              global tcp= get_actual_tcp_pose ()
              $ 1343 "offset_altura≔p[tcp[0],tcp[1],((alta-0.0095)-(acomodo/1000)),tcp[3],tcp[4],tcp[5]]"
              global offset_altura=p[tcp[0],tcp[1],((alta-0.0095)-(acomodo/1000)),tcp[3],tcp[4],tcp[5]]
              $ 1344 "MoveL"
              $ 1345 "offset_altura" "breakAfter"
              movel(offset_altura, a=0.04, v=0.03)
            end
            $ 1346 "Freemove"
            $ 1347 "Wait: 2.0"
            sleep(2.0)
            $ 1348 "freedrive_mode()"
            freedrive_mode()
            $ 1349 "Wait: 2.5"
            sleep(2.5)
            $ 1350 "end_freedrive_mode()"
            end_freedrive_mode()
            $ 1351 "Wait: 0.3"
            sleep(0.3)
            $ 1352 "Set CO[1]=Encender"
            set_configurable_digital_out(1, True)
            $ 1353 "Wait: 1.0"
            sleep(1.0)
            $ 1354 "Wait: 0.3"
            sleep(0.3)
            $ 1355 "Wait: 0.3"
            sleep(0.3)
            $ 1356 "Wait: 0.3"
            sleep(0.3)
            $ 1357 "Loop 2 times"
            Loop_50 = 0
            while (Loop_50 < 2):
              $ 1358 "Poses_taladrado≔pose_sub(get_actual_tcp_pose(), bajada_broca)"
              global Poses_taladrado= pose_sub ( get_actual_tcp_pose (), bajada_broca)
              $ 1359 "Poses_taladrado" "breakAfter"
              movel(Poses_taladrado, a=0.005, v=0.001)
              $ 1360 "If bajada_broca≟p[0,0,0.018,0,0,0]"
              if (bajada_broca == p[0,0,0.018,0,0,0]):
                $ 1361 "num_barreno≔str_cat('Barreno: ',barrenoActual)"
                global num_barreno=str_cat("Barreno: ",barrenoActual)
                $ 1362 "tcp_actual≔get_actual_tcp_pose()"
                global tcp_actual= get_actual_tcp_pose ()
                $ 1363 "X_actual≔str_cat('     X: ',tcp_actual[0])"
                global X_actual=str_cat("     X: ",tcp_actual[0])
                $ 1364 "Y_actual≔str_cat('     Y: ',tcp_actual[1])"
                global Y_actual=str_cat("     Y: ",tcp_actual[1])
                $ 1365 "pos_barreno≔str_cat(X_actual,Y_actual)"
                global pos_barreno=str_cat(X_actual,Y_actual)
                $ 1366 "textmsg(num_barreno,pos_barreno)"
                textmsg(num_barreno,pos_barreno)
              end
              $ 1367 "Poses_taladrado≔pose_add(get_actual_tcp_pose(), bajada_broca)"
              global Poses_taladrado= pose_add ( get_actual_tcp_pose (), bajada_broca)
              $ 1368 "Poses_taladrado" "breakAfter"
              movel(Poses_taladrado, a=0.01, v=0.01)
              $ 1369 "bajada_broca≔pose_add(bajada_broca, p[0,0,0.009,0,0,0])"
              global bajada_broca= pose_add (bajada_broca, p[0,0,0.009,0,0,0])
              Loop_50 = Loop_50 + 1
            end
            $ 1370 "Direction: Base Z+"
            global move_thread_flag_1370=0
            thread move_thread_1370():
              enter_critical
              move_thread_flag_1370 = 1
              local towardsPos=calculate_point_to_move_towards(p[0.0,0.0,0.0,0.0,0.0,0.0], [0.0,0.0,1.0], 0.05)
              movel(towardsPos, a=0.01, v=0.01)
              move_thread_flag_1370 = 2
              exit_critical
            end
            move_thread_flag_1370 = 0
            move_thread_han_1370 = run move_thread_1370()
            while (True):
              sleep(1.0E-10)
              if (move_thread_flag_1370 > 1):
                join move_thread_han_1370
                $ 1371 "Until (distance)"
                break
              end
              sync()
            end
            $ 1372 "MoveJ"
            $ 1373 "internos" "breakAfter"
            movej(internos, a=0.6981317007977318, v=0.5235987755982988)
            $ 1374 "Wait: 0.3"
            sleep(0.3)
            $ 1375 "Set CO[1]=Apagar"
            set_configurable_digital_out(1, False)
            $ 1376 "Wait: 0.3"
            sleep(0.3)
            $ 1377 "If barrenoActual≟13 or barrenoActual≟27"
            if (barrenoActual == 13  or  barrenoActual == 27):
              $ 1378 "Direction: Base Z+"
              global move_thread_flag_1378=0
              thread move_thread_1378():
                enter_critical
                move_thread_flag_1378 = 1
                local towardsPos=calculate_point_to_move_towards(p[0.0,0.0,0.0,0.0,0.0,0.0], [0.0,0.0,1.0], 0.03)
                movel(towardsPos, a=0.04, v=0.03)
                move_thread_flag_1378 = 2
                exit_critical
              end
              move_thread_flag_1378 = 0
              move_thread_han_1378 = run move_thread_1378()
              while (True):
                sleep(1.0E-10)
                if (move_thread_flag_1378 > 1):
                  join move_thread_han_1378
                  $ 1379 "Until (distance)"
                  break
                end
                sync()
              end
              $ 1380 "MoveJ"
              $ 1381 "Zona_der1" "breakAfter"
              movej(get_inverse_kin(Zona_der1_p, qnear=Zona_der1_q), a=0.6981317007977318, v=0.5235987755982988)
              $ 1382 "Posicion_Cero" "breakAfter"
              movej(get_inverse_kin(Posicion_Cero_p, qnear=Posicion_Cero_q), a=0.6981317007977318, v=0.5235987755982988)
              $ 1383 "Call Quitar_Broca_Chida"
              Quitar_Broca_Chida()
              $ 1384 "If barrenoActual≟13"
              if (barrenoActual == 13):
                $ 1385 "Call Poner_Broca"
                Poner_Broca()
              else:
                $ 1386 "ElseIf barrenoActual≟27"
                if (barrenoActual == 27):
                  $ 1387 "Call Poner_Broca"
                  Poner_Broca()
                end
              end
              $ 1388 "MoveJ"
              $ 1389 "Posicion_Cero" "breakAfter"
              movej(get_inverse_kin(Posicion_Cero_p, qnear=Posicion_Cero_q), a=0.6981317007977318, v=0.5235987755982988)
              $ 1390 "Zona_der1" "breakAfter"
              movej(get_inverse_kin(Zona_der1_p, qnear=Zona_der1_q), a=0.6981317007977318, v=0.5235987755982988)
            end
            $ 1391 "barrenoActual≔barrenoActual+1"
            global barrenoActual=barrenoActual+1
          end
          $ 1392 "Linea 2 a 1935"
          $ 1393 "broca≔1935"
          global broca=1935
          $ 1394 "Buje_inicial"
          $ 1395 "Buje_Inicial≔L2B2"
          global Buje_Inicial=L2B2
          $ 1396 "Buje_final"
          $ 1397 "Buje_Final≔L2B1"
          global Buje_Final=L2B1
          $ 1398 "barrenosTotales≔27"
          global barrenosTotales=27
          $ 1399 "barrenoActual≔1"
          global barrenoActual=1
          $ 1400 "Loop barrenoActual≤barrenosTotales"
          while (barrenoActual <= barrenosTotales):
            $ 1401 "MoveL"
            $ 1402 "bajada_broca≔p[0,0,0.009,0,0,0]"
            global bajada_broca=p[0,0,0.009,0,0,0]
            $ 1403 "internos≔interpolate_pose(Buje_Inicial, Buje_Final, ((barrenoActual)-1)/((barrenosTotales)-1))"
            global internos= interpolate_pose (Buje_Inicial, Buje_Final, ((barrenoActual)-1)/((barrenosTotales)-1))
            $ 1404 "Alturas"
            $ 1405 "If barrenoActual≟1 or barrenoActual≟3 or barrenoActual≟5 or barrenoActual≟7 or barrenoActual≟9 or barrenoActual≟11 or barrenoActual≟13 or barrenoActual≟15 or barrenoActual≟17 or barrenoActual≟19 or barrenoActual≟21 or barrenoActual≟23 or barrenoActual≟25 or barrenoActual≟27"
            if (barrenoActual == 1  or  barrenoActual == 3  or  barrenoActual == 5  or  barrenoActual == 7  or  barrenoActual == 9  or  barrenoActual == 11  or  barrenoActual == 13  or  barrenoActual == 15  or  barrenoActual == 17  or  barrenoActual == 19  or  barrenoActual == 21  or  barrenoActual == 23  or  barrenoActual == 25  or  barrenoActual == 27):
              $ 1406 "Set mensaje_mw10=200"
              modbus_set_output_register("mensaje_mw10", 200)
              $ 1407 "Wait Continuar_M30=HI"
              while (modbus_get_signal_status("Continuar_M30") == False):
                sync()
              end
              $ 1408 "Wait: 1.0"
              sleep(1.0)
              $ 1409 "Set mensaje_mw10=150"
              modbus_set_output_register("mensaje_mw10", 150)
              $ 1410 "Wait: 1.0"
              sleep(1.0)
            end
            $ 1411 "MoveJ"
            $ 1412 "internos" "breakAfter"
            movej(internos, a=0.6981317007977318, v=0.5235987755982988)
            $ 1413 "Wait: 2.0"
            sleep(2.0)
            $ 1414 "If P1h[2]<P2h[2]"
            if (P1h[2]<P2h[2]):
              $ 1415 "acomodo≔(altura/(barrenosTotales-1))*(barrenoActual-1)"
              global acomodo=(altura/(barrenosTotales-1))*(barrenoActual-1)
              $ 1416 "tcp≔get_actual_tcp_pose()"
              global tcp= get_actual_tcp_pose ()
              $ 1417 "offset_altura≔p[tcp[0],tcp[1],((alta-0.0095)-(acomodo/1000)),tcp[3],tcp[4],tcp[5]]"
              global offset_altura=p[tcp[0],tcp[1],((alta-0.0095)-(acomodo/1000)),tcp[3],tcp[4],tcp[5]]
              $ 1418 "MoveL"
              $ 1419 "offset_altura" "breakAfter"
              movel(offset_altura, a=0.04, v=0.03)
            else:
              $ 1420 "Else" "noBreak"
              $ 1421 "acomodo≔(altura/(barrenosTotales-1))*(26-(barrenoActual-1))"
              global acomodo=(altura/(barrenosTotales-1))*(26-(barrenoActual-1))
              $ 1422 "tcp≔get_actual_tcp_pose()"
              global tcp= get_actual_tcp_pose ()
              $ 1423 "offset_altura≔p[tcp[0],tcp[1],((alta-0.0095)-(acomodo/1000)),tcp[3],tcp[4],tcp[5]]"
              global offset_altura=p[tcp[0],tcp[1],((alta-0.0095)-(acomodo/1000)),tcp[3],tcp[4],tcp[5]]
              $ 1424 "MoveL"
              $ 1425 "offset_altura" "breakAfter"
              movel(offset_altura, a=0.04, v=0.03)
            end
            $ 1426 "Freemove"
            $ 1427 "Wait: 2.0"
            sleep(2.0)
            $ 1428 "freedrive_mode()"
            freedrive_mode()
            $ 1429 "Wait: 2.5"
            sleep(2.5)
            $ 1430 "end_freedrive_mode()"
            end_freedrive_mode()
            $ 1431 "Wait: 0.3"
            sleep(0.3)
            $ 1432 "Set CO[1]=Encender"
            set_configurable_digital_out(1, True)
            $ 1433 "Wait: 1.0"
            sleep(1.0)
            $ 1434 "Wait: 0.3"
            sleep(0.3)
            $ 1435 "Wait: 0.3"
            sleep(0.3)
            $ 1436 "Wait: 0.3"
            sleep(0.3)
            $ 1437 "Loop 2 times"
            Loop_54 = 0
            while (Loop_54 < 2):
              $ 1438 "Poses_taladrado≔pose_sub(get_actual_tcp_pose(), bajada_broca)"
              global Poses_taladrado= pose_sub ( get_actual_tcp_pose (), bajada_broca)
              $ 1439 "Poses_taladrado" "breakAfter"
              movel(Poses_taladrado, a=0.005, v=0.001)
              $ 1440 "If bajada_broca≟p[0,0,0.018,0,0,0]"
              if (bajada_broca == p[0,0,0.018,0,0,0]):
                $ 1441 "num_barreno≔str_cat('Barreno: ',barrenoActual)"
                global num_barreno=str_cat("Barreno: ",barrenoActual)
                $ 1442 "tcp_actual≔get_actual_tcp_pose()"
                global tcp_actual= get_actual_tcp_pose ()
                $ 1443 "X_actual≔str_cat('     X: ',tcp_actual[0])"
                global X_actual=str_cat("     X: ",tcp_actual[0])
                $ 1444 "Y_actual≔str_cat('     Y: ',tcp_actual[1])"
                global Y_actual=str_cat("     Y: ",tcp_actual[1])
                $ 1445 "pos_barreno≔str_cat(X_actual,Y_actual)"
                global pos_barreno=str_cat(X_actual,Y_actual)
                $ 1446 "textmsg(num_barreno,pos_barreno)"
                textmsg(num_barreno,pos_barreno)
              end
              $ 1447 "Poses_taladrado≔pose_add(get_actual_tcp_pose(), bajada_broca)"
              global Poses_taladrado= pose_add ( get_actual_tcp_pose (), bajada_broca)
              $ 1448 "Poses_taladrado" "breakAfter"
              movel(Poses_taladrado, a=0.01, v=0.01)
              $ 1449 "bajada_broca≔pose_add(bajada_broca, p[0,0,0.009,0,0,0])"
              global bajada_broca= pose_add (bajada_broca, p[0,0,0.009,0,0,0])
              Loop_54 = Loop_54 + 1
            end
            $ 1450 "Direction: Base Z+"
            global move_thread_flag_1450=0
            thread move_thread_1450():
              enter_critical
              move_thread_flag_1450 = 1
              local towardsPos=calculate_point_to_move_towards(p[0.0,0.0,0.0,0.0,0.0,0.0], [0.0,0.0,1.0], 0.05)
              movel(towardsPos, a=0.01, v=0.01)
              move_thread_flag_1450 = 2
              exit_critical
            end
            move_thread_flag_1450 = 0
            move_thread_han_1450 = run move_thread_1450()
            while (True):
              sleep(1.0E-10)
              if (move_thread_flag_1450 > 1):
                join move_thread_han_1450
                $ 1451 "Until (distance)"
                break
              end
              sync()
            end
            $ 1452 "MoveJ"
            $ 1453 "internos" "breakAfter"
            movej(internos, a=0.6981317007977318, v=0.5235987755982988)
            $ 1454 "Wait: 0.3"
            sleep(0.3)
            $ 1455 "Set CO[1]=Apagar"
            set_configurable_digital_out(1, False)
            $ 1456 "Wait: 0.3"
            sleep(0.3)
            $ 1457 "If barrenoActual≟13"
            if (barrenoActual == 13):
              $ 1458 "Direction: Base Z+"
              global move_thread_flag_1458=0
              thread move_thread_1458():
                enter_critical
                move_thread_flag_1458 = 1
                local towardsPos=calculate_point_to_move_towards(p[0.0,0.0,0.0,0.0,0.0,0.0], [0.0,0.0,1.0], 0.03)
                movel(towardsPos, a=0.04, v=0.03)
                move_thread_flag_1458 = 2
                exit_critical
              end
              move_thread_flag_1458 = 0
              move_thread_han_1458 = run move_thread_1458()
              while (True):
                sleep(1.0E-10)
                if (move_thread_flag_1458 > 1):
                  join move_thread_han_1458
                  $ 1459 "Until (distance)"
                  break
                end
                sync()
              end
              $ 1460 "MoveJ"
              $ 1461 "Zona_der1" "breakAfter"
              movej(get_inverse_kin(Zona_der1_p, qnear=Zona_der1_q), a=1.3962634015954636, v=1.0471975511965976)
              $ 1462 "Posicion_Cero" "breakAfter"
              movej(get_inverse_kin(Posicion_Cero_p, qnear=Posicion_Cero_q), a=1.3962634015954636, v=1.0471975511965976)
              $ 1463 "Call Quitar_Broca_Chida"
              Quitar_Broca_Chida()
              $ 1464 "Call Poner_Broca"
              Poner_Broca()
              $ 1465 "MoveJ"
              $ 1466 "Posicion_Cero" "breakAfter"
              movej(get_inverse_kin(Posicion_Cero_p, qnear=Posicion_Cero_q), a=1.3962634015954636, v=1.0471975511965976)
              $ 1467 "Zona_der1" "breakAfter"
              movej(get_inverse_kin(Zona_der1_p, qnear=Zona_der1_q), a=1.3962634015954636, v=1.0471975511965976)
            else:
              $ 1468 "ElseIf barrenoActual≟27"
              if (barrenoActual == 27):
                $ 1469 "Direction: Base Z+"
                global move_thread_flag_1469=0
                thread move_thread_1469():
                  enter_critical
                  move_thread_flag_1469 = 1
                  local towardsPos=calculate_point_to_move_towards(p[0.0,0.0,0.0,0.0,0.0,0.0], [0.0,0.0,1.0], 0.03)
                  movel(towardsPos, a=0.04, v=0.03)
                  move_thread_flag_1469 = 2
                  exit_critical
                end
                move_thread_flag_1469 = 0
                move_thread_han_1469 = run move_thread_1469()
                while (True):
                  sleep(1.0E-10)
                  if (move_thread_flag_1469 > 1):
                    join move_thread_han_1469
                    $ 1470 "Until (distance)"
                    break
                  end
                  sync()
                end
                $ 1471 "MoveJ"
                $ 1472 "Zona_der1" "breakAfter"
                movej(get_inverse_kin(Zona_der1_p, qnear=Zona_der1_q), a=1.3962634015954636, v=1.0471975511965976)
                $ 1473 "Posicion_Cero" "breakAfter"
                movej(get_inverse_kin(Posicion_Cero_p, qnear=Posicion_Cero_q), a=1.3962634015954636, v=1.0471975511965976)
                $ 1474 "Call Quitar_Broca_Chida"
                Quitar_Broca_Chida()
                $ 1475 "Set carrusel_home=Encender"
                modbus_set_output_signal("carrusel_home", True)
                $ 1476 "Wait: 1.0"
                sleep(1.0)
                $ 1477 "Set carrusel_home=Apagar"
                modbus_set_output_signal("carrusel_home", False)
                $ 1478 "Set mensaje_mw10=85"
                modbus_set_output_register("mensaje_mw10", 85)
                $ 1479 "Wait Continuar_M30=HI"
                while (modbus_get_signal_status("Continuar_M30") == False):
                  sync()
                end
                $ 1480 "Wait: 1.0"
                sleep(1.0)
                $ 1481 "Set mensaje_mw10=120"
                modbus_set_output_register("mensaje_mw10", 120)
                $ 1482 "Wait Continuar_M30=HI"
                while (modbus_get_signal_status("Continuar_M30") == False):
                  sync()
                end
                $ 1483 "Wait: 1.0"
                sleep(1.0)
                $ 1484 "Set carrusel_home=Encender"
                modbus_set_output_signal("carrusel_home", True)
                $ 1485 "Wait: 1.0"
                sleep(1.0)
                $ 1486 "Set carrusel_home=Apagar"
                modbus_set_output_signal("carrusel_home", False)
                $ 1487 "Set mensaje_mw10=90"
                modbus_set_output_register("mensaje_mw10", 90)
                $ 1488 "Wait Continuar_M30=HI"
                while (modbus_get_signal_status("Continuar_M30") == False):
                  sync()
                end
                $ 1489 "Wait: 1.0"
                sleep(1.0)
                $ 1490 "Call Poner_Broca"
                Poner_Broca()
                $ 1491 "broca≔217"
                global broca=217
                $ 1492 "MoveJ"
                $ 1493 "Posicion_Cero" "breakAfter"
                movej(get_inverse_kin(Posicion_Cero_p, qnear=Posicion_Cero_q), a=1.3962634015954636, v=1.0471975511965976)
                $ 1494 "Zona_der1" "breakAfter"
                movej(get_inverse_kin(Zona_der1_p, qnear=Zona_der1_q), a=1.3962634015954636, v=1.0471975511965976)
                $ 1495 "Set mensaje_mw10=95"
                modbus_set_output_register("mensaje_mw10", 95)
                $ 1496 "Wait Continuar_M30=HI"
                while (modbus_get_signal_status("Continuar_M30") == False):
                  sync()
                end
                $ 1497 "Wait: 1.0"
                sleep(1.0)
                $ 1498 "Set mensaje_mw10=150"
                modbus_set_output_register("mensaje_mw10", 150)
                $ 1499 "Wait Continuar_M30=HI"
                while (modbus_get_signal_status("Continuar_M30") == False):
                  sync()
                end
                $ 1500 "Wait: 1.0"
                sleep(1.0)
              end
            end
            $ 1501 "barrenoActual≔barrenoActual+1"
            global barrenoActual=barrenoActual+1
          end
          $ 1502 "Linea 1 a 217"
          $ 1503 "broca≔217"
          global broca=217
          $ 1504 "Buje_inicial"
          $ 1505 "Buje_Inicial≔L1B2"
          global Buje_Inicial=L1B2
          $ 1506 "Buje_final"
          $ 1507 "Buje_Final≔L1B1"
          global Buje_Final=L1B1
          $ 1508 "barrenosTotales≔27"
          global barrenosTotales=27
          $ 1509 "barrenoActual≔1"
          global barrenoActual=1
          $ 1510 "Loop barrenoActual≤barrenosTotales"
          while (barrenoActual <= barrenosTotales):
            $ 1511 "MoveL"
            $ 1512 "bajada_broca≔p[0,0,0.018,0,0,0]"
            global bajada_broca=p[0,0,0.018,0,0,0]
            $ 1513 "internos≔interpolate_pose(Buje_Inicial, Buje_Final, ((barrenoActual)-1)/((barrenosTotales)-1))"
            global internos= interpolate_pose (Buje_Inicial, Buje_Final, ((barrenoActual)-1)/((barrenosTotales)-1))
            $ 1514 "Wait: 2.0"
            sleep(2.0)
            $ 1515 "Alturas"
            $ 1516 "If barrenoActual≟1 or barrenoActual≟3 or barrenoActual≟5 or barrenoActual≟7 or barrenoActual≟9 or barrenoActual≟11 or barrenoActual≟13 or barrenoActual≟15 or barrenoActual≟17 or barrenoActual≟19 or barrenoActual≟21 or barrenoActual≟23 or barrenoActual≟25 or barrenoActual≟27"
            if (barrenoActual == 1  or  barrenoActual == 3  or  barrenoActual == 5  or  barrenoActual == 7  or  barrenoActual == 9  or  barrenoActual == 11  or  barrenoActual == 13  or  barrenoActual == 15  or  barrenoActual == 17  or  barrenoActual == 19  or  barrenoActual == 21  or  barrenoActual == 23  or  barrenoActual == 25  or  barrenoActual == 27):
              $ 1517 "Set mensaje_mw10=200"
              modbus_set_output_register("mensaje_mw10", 200)
              $ 1518 "Wait Continuar_M30=HI"
              while (modbus_get_signal_status("Continuar_M30") == False):
                sync()
              end
              $ 1519 "Wait: 1.0"
              sleep(1.0)
              $ 1520 "Set mensaje_mw10=150"
              modbus_set_output_register("mensaje_mw10", 150)
              $ 1521 "Wait: 1.0"
              sleep(1.0)
            end
            $ 1522 "MoveJ"
            $ 1523 "internos" "breakAfter"
            movej(internos, a=0.6981317007977318, v=0.5235987755982988)
            $ 1524 "Wait: 2.0"
            sleep(2.0)
            $ 1525 "If P1h[2]<P2h[2]"
            if (P1h[2]<P2h[2]):
              $ 1526 "acomodo≔(altura/(barrenosTotales-1))*(barrenoActual-1)"
              global acomodo=(altura/(barrenosTotales-1))*(barrenoActual-1)
              $ 1527 "tcp≔get_actual_tcp_pose()"
              global tcp= get_actual_tcp_pose ()
              $ 1528 "offset_altura≔p[tcp[0],tcp[1],((alta-0.0095)-(acomodo/1000)),tcp[3],tcp[4],tcp[5]]"
              global offset_altura=p[tcp[0],tcp[1],((alta-0.0095)-(acomodo/1000)),tcp[3],tcp[4],tcp[5]]
              $ 1529 "MoveL"
              $ 1530 "offset_altura" "breakAfter"
              movel(offset_altura, a=0.04, v=0.03)
            else:
              $ 1531 "Else" "noBreak"
              $ 1532 "acomodo≔(altura/(barrenosTotales-1))*(26-(barrenoActual-1))"
              global acomodo=(altura/(barrenosTotales-1))*(26-(barrenoActual-1))
              $ 1533 "tcp≔get_actual_tcp_pose()"
              global tcp= get_actual_tcp_pose ()
              $ 1534 "offset_altura≔p[tcp[0],tcp[1],((alta-0.0095)-(acomodo/1000)),tcp[3],tcp[4],tcp[5]]"
              global offset_altura=p[tcp[0],tcp[1],((alta-0.0095)-(acomodo/1000)),tcp[3],tcp[4],tcp[5]]
              $ 1535 "MoveL"
              $ 1536 "offset_altura" "breakAfter"
              movel(offset_altura, a=0.04, v=0.03)
            end
            $ 1537 "Freemove"
            $ 1538 "Wait: 2.0"
            sleep(2.0)
            $ 1539 "freedrive_mode()"
            freedrive_mode()
            $ 1540 "Wait: 2.5"
            sleep(2.5)
            $ 1541 "end_freedrive_mode()"
            end_freedrive_mode()
            $ 1542 "Wait: 0.3"
            sleep(0.3)
            $ 1543 "Set CO[1]=Encender"
            set_configurable_digital_out(1, True)
            $ 1544 "Wait: 1.0"
            sleep(1.0)
            $ 1545 "Wait: 0.3"
            sleep(0.3)
            $ 1546 "Wait: 0.3"
            sleep(0.3)
            $ 1547 "Wait: 0.3"
            sleep(0.3)
            $ 1548 "Loop 1 times"
            Loop_56 = 0
            while (Loop_56 < 1):
              $ 1549 "Poses_taladrado≔pose_sub(get_actual_tcp_pose(), bajada_broca)"
              global Poses_taladrado= pose_sub ( get_actual_tcp_pose (), bajada_broca)
              $ 1550 "Poses_taladrado" "breakAfter"
              movel(Poses_taladrado, a=0.005, v=0.001)
              $ 1551 "If bajada_broca≟p[0,0,0.018,0,0,0]"
              if (bajada_broca == p[0,0,0.018,0,0,0]):
                $ 1552 "num_barreno≔str_cat('Barreno: ',barrenoActual)"
                global num_barreno=str_cat("Barreno: ",barrenoActual)
                $ 1553 "tcp_actual≔get_actual_tcp_pose()"
                global tcp_actual= get_actual_tcp_pose ()
                $ 1554 "X_actual≔str_cat('     X: ',tcp_actual[0])"
                global X_actual=str_cat("     X: ",tcp_actual[0])
                $ 1555 "Y_actual≔str_cat('     Y: ',tcp_actual[1])"
                global Y_actual=str_cat("     Y: ",tcp_actual[1])
                $ 1556 "pos_barreno≔str_cat(X_actual,Y_actual)"
                global pos_barreno=str_cat(X_actual,Y_actual)
                $ 1557 "textmsg(num_barreno,pos_barreno)"
                textmsg(num_barreno,pos_barreno)
              end
              $ 1558 "Poses_taladrado≔pose_add(get_actual_tcp_pose(), bajada_broca)"
              global Poses_taladrado= pose_add ( get_actual_tcp_pose (), bajada_broca)
              $ 1559 "Poses_taladrado" "breakAfter"
              movel(Poses_taladrado, a=0.01, v=0.01)
              $ 1560 "bajada_broca≔pose_add(bajada_broca, p[0,0,0.018,0,0,0])"
              global bajada_broca= pose_add (bajada_broca, p[0,0,0.018,0,0,0])
              Loop_56 = Loop_56 + 1
            end
            $ 1561 "Direction: Base Z+"
            global move_thread_flag_1561=0
            thread move_thread_1561():
              enter_critical
              move_thread_flag_1561 = 1
              local towardsPos=calculate_point_to_move_towards(p[0.0,0.0,0.0,0.0,0.0,0.0], [0.0,0.0,1.0], 0.05)
              movel(towardsPos, a=0.01, v=0.01)
              move_thread_flag_1561 = 2
              exit_critical
            end
            move_thread_flag_1561 = 0
            move_thread_han_1561 = run move_thread_1561()
            while (True):
              sleep(1.0E-10)
              if (move_thread_flag_1561 > 1):
                join move_thread_han_1561
                $ 1562 "Until (distance)"
                break
              end
              sync()
            end
            $ 1563 "MoveJ"
            $ 1564 "internos" "breakAfter"
            movej(internos, a=0.6981317007977318, v=0.5235987755982988)
            $ 1565 "Wait: 0.3"
            sleep(0.3)
            $ 1566 "Set CO[1]=Apagar"
            set_configurable_digital_out(1, False)
            $ 1567 "Wait: 0.3"
            sleep(0.3)
            $ 1568 "If barrenoActual≟13 or barrenoActual≟27"
            if (barrenoActual == 13  or  barrenoActual == 27):
              $ 1569 "Direction: Base Z+"
              global move_thread_flag_1569=0
              thread move_thread_1569():
                enter_critical
                move_thread_flag_1569 = 1
                local towardsPos=calculate_point_to_move_towards(p[0.0,0.0,0.0,0.0,0.0,0.0], [0.0,0.0,1.0], 0.03)
                movel(towardsPos, a=0.03, v=0.04)
                move_thread_flag_1569 = 2
                exit_critical
              end
              move_thread_flag_1569 = 0
              move_thread_han_1569 = run move_thread_1569()
              while (True):
                sleep(1.0E-10)
                if (move_thread_flag_1569 > 1):
                  join move_thread_han_1569
                  $ 1570 "Until (distance)"
                  break
                end
                sync()
              end
              $ 1571 "MoveJ"
              $ 1572 "Zona_der1" "breakAfter"
              movej(get_inverse_kin(Zona_der1_p, qnear=Zona_der1_q), a=0.6981317007977318, v=0.5235987755982988)
              $ 1573 "Posicion_Cero" "breakAfter"
              movej(get_inverse_kin(Posicion_Cero_p, qnear=Posicion_Cero_q), a=0.6981317007977318, v=0.5235987755982988)
              $ 1574 "Call Quitar_Broca_Chida"
              Quitar_Broca_Chida()
              $ 1575 "If barrenoActual≟13"
              if (barrenoActual == 13):
                $ 1576 "Call Poner_Broca"
                Poner_Broca()
              else:
                $ 1577 "ElseIf barrenoActual≟27"
                if (barrenoActual == 27):
                  $ 1578 "Call Poner_Broca"
                  Poner_Broca()
                end
              end
              $ 1579 "MoveJ"
              $ 1580 "Posicion_Cero" "breakAfter"
              movej(get_inverse_kin(Posicion_Cero_p, qnear=Posicion_Cero_q), a=0.6981317007977318, v=0.5235987755982988)
              $ 1581 "Zona_der1" "breakAfter"
              movej(get_inverse_kin(Zona_der1_p, qnear=Zona_der1_q), a=0.6981317007977318, v=0.5235987755982988)
            end
            $ 1582 "barrenoActual≔barrenoActual+1"
            global barrenoActual=barrenoActual+1
          end
          $ 1583 "Linea 2 a 217"
          $ 1584 "broca≔217"
          global broca=217
          $ 1585 "Buje_inicial"
          $ 1586 "Buje_Inicial≔L2B2"
          global Buje_Inicial=L2B2
          $ 1587 "Buje_final"
          $ 1588 "Buje_Final≔L2B1"
          global Buje_Final=L2B1
          $ 1589 "barrenosTotales≔27"
          global barrenosTotales=27
          $ 1590 "barrenoActual≔1"
          global barrenoActual=1
          $ 1591 "Loop barrenoActual≤barrenosTotales"
          while (barrenoActual <= barrenosTotales):
            $ 1592 "MoveL"
            $ 1593 "bajada_broca≔p[0,0,0.018,0,0,0]"
            global bajada_broca=p[0,0,0.018,0,0,0]
            $ 1594 "internos≔interpolate_pose(Buje_Inicial, Buje_Final, ((barrenoActual)-1)/((barrenosTotales)-1))"
            global internos= interpolate_pose (Buje_Inicial, Buje_Final, ((barrenoActual)-1)/((barrenosTotales)-1))
            $ 1595 "Alturas"
            $ 1596 "If barrenoActual≟1 or barrenoActual≟3 or barrenoActual≟5 or barrenoActual≟7 or barrenoActual≟9 or barrenoActual≟11 or barrenoActual≟13 or barrenoActual≟15 or barrenoActual≟17 or barrenoActual≟19 or barrenoActual≟21 or barrenoActual≟23 or barrenoActual≟25 or barrenoActual≟27"
            if (barrenoActual == 1  or  barrenoActual == 3  or  barrenoActual == 5  or  barrenoActual == 7  or  barrenoActual == 9  or  barrenoActual == 11  or  barrenoActual == 13  or  barrenoActual == 15  or  barrenoActual == 17  or  barrenoActual == 19  or  barrenoActual == 21  or  barrenoActual == 23  or  barrenoActual == 25  or  barrenoActual == 27):
              $ 1597 "Set mensaje_mw10=200"
              modbus_set_output_register("mensaje_mw10", 200)
              $ 1598 "Wait Continuar_M30=HI"
              while (modbus_get_signal_status("Continuar_M30") == False):
                sync()
              end
              $ 1599 "Wait: 1.0"
              sleep(1.0)
              $ 1600 "Set mensaje_mw10=150"
              modbus_set_output_register("mensaje_mw10", 150)
              $ 1601 "Wait: 1.0"
              sleep(1.0)
            end
            $ 1602 "MoveJ"
            $ 1603 "internos" "breakAfter"
            movej(internos, a=0.6981317007977318, v=0.5235987755982988)
            $ 1604 "Wait: 2.0"
            sleep(2.0)
            $ 1605 "If P1h[2]<P2h[2]"
            if (P1h[2]<P2h[2]):
              $ 1606 "acomodo≔(altura/(barrenosTotales-1))*(barrenoActual-1)"
              global acomodo=(altura/(barrenosTotales-1))*(barrenoActual-1)
              $ 1607 "tcp≔get_actual_tcp_pose()"
              global tcp= get_actual_tcp_pose ()
              $ 1608 "offset_altura≔p[tcp[0],tcp[1],((alta-0.0095)-(acomodo/1000)),tcp[3],tcp[4],tcp[5]]"
              global offset_altura=p[tcp[0],tcp[1],((alta-0.0095)-(acomodo/1000)),tcp[3],tcp[4],tcp[5]]
              $ 1609 "MoveL"
              $ 1610 "offset_altura" "breakAfter"
              movel(offset_altura, a=0.04, v=0.03)
            else:
              $ 1611 "Else" "noBreak"
              $ 1612 "acomodo≔(altura/(barrenosTotales-1))*(26-(barrenoActual-1))"
              global acomodo=(altura/(barrenosTotales-1))*(26-(barrenoActual-1))
              $ 1613 "tcp≔get_actual_tcp_pose()"
              global tcp= get_actual_tcp_pose ()
              $ 1614 "offset_altura≔p[tcp[0],tcp[1],((alta-0.0095)-(acomodo/1000)),tcp[3],tcp[4],tcp[5]]"
              global offset_altura=p[tcp[0],tcp[1],((alta-0.0095)-(acomodo/1000)),tcp[3],tcp[4],tcp[5]]
              $ 1615 "MoveL"
              $ 1616 "offset_altura" "breakAfter"
              movel(offset_altura, a=0.04, v=0.03)
            end
            $ 1617 "Freemove"
            $ 1618 "Wait: 2.0"
            sleep(2.0)
            $ 1619 "freedrive_mode()"
            freedrive_mode()
            $ 1620 "Wait: 2.5"
            sleep(2.5)
            $ 1621 "end_freedrive_mode()"
            end_freedrive_mode()
            $ 1622 "Wait: 0.3"
            sleep(0.3)
            $ 1623 "Set CO[1]=Encender"
            set_configurable_digital_out(1, True)
            $ 1624 "Wait: 1.0"
            sleep(1.0)
            $ 1625 "Wait: 0.3"
            sleep(0.3)
            $ 1626 "Wait: 0.3"
            sleep(0.3)
            $ 1627 "Wait: 0.3"
            sleep(0.3)
            $ 1628 "Loop 1 times"
            Loop_58 = 0
            while (Loop_58 < 1):
              $ 1629 "Poses_taladrado≔pose_sub(get_actual_tcp_pose(), bajada_broca)"
              global Poses_taladrado= pose_sub ( get_actual_tcp_pose (), bajada_broca)
              $ 1630 "Poses_taladrado" "breakAfter"
              movel(Poses_taladrado, a=0.005, v=0.001)
              $ 1631 "If bajada_broca≟p[0,0,0.018,0,0,0]"
              if (bajada_broca == p[0,0,0.018,0,0,0]):
                $ 1632 "num_barreno≔str_cat('Barreno: ',barrenoActual)"
                global num_barreno=str_cat("Barreno: ",barrenoActual)
                $ 1633 "tcp_actual≔get_actual_tcp_pose()"
                global tcp_actual= get_actual_tcp_pose ()
                $ 1634 "X_actual≔str_cat('     X: ',tcp_actual[0])"
                global X_actual=str_cat("     X: ",tcp_actual[0])
                $ 1635 "Y_actual≔str_cat('     Y: ',tcp_actual[1])"
                global Y_actual=str_cat("     Y: ",tcp_actual[1])
                $ 1636 "pos_barreno≔str_cat(X_actual,Y_actual)"
                global pos_barreno=str_cat(X_actual,Y_actual)
                $ 1637 "textmsg(num_barreno,pos_barreno)"
                textmsg(num_barreno,pos_barreno)
              end
              $ 1638 "Poses_taladrado≔pose_add(get_actual_tcp_pose(), bajada_broca)"
              global Poses_taladrado= pose_add ( get_actual_tcp_pose (), bajada_broca)
              $ 1639 "Poses_taladrado" "breakAfter"
              movel(Poses_taladrado, a=0.01, v=0.01)
              $ 1640 "bajada_broca≔pose_add(bajada_broca, p[0,0,0.018,0,0,0])"
              global bajada_broca= pose_add (bajada_broca, p[0,0,0.018,0,0,0])
              Loop_58 = Loop_58 + 1
            end
            $ 1641 "Direction: Base Z+"
            global move_thread_flag_1641=0
            thread move_thread_1641():
              enter_critical
              move_thread_flag_1641 = 1
              local towardsPos=calculate_point_to_move_towards(p[0.0,0.0,0.0,0.0,0.0,0.0], [0.0,0.0,1.0], 0.05)
              movel(towardsPos, a=0.01, v=0.01)
              move_thread_flag_1641 = 2
              exit_critical
            end
            move_thread_flag_1641 = 0
            move_thread_han_1641 = run move_thread_1641()
            while (True):
              sleep(1.0E-10)
              if (move_thread_flag_1641 > 1):
                join move_thread_han_1641
                $ 1642 "Until (distance)"
                break
              end
              sync()
            end
            $ 1643 "MoveJ"
            $ 1644 "internos" "breakAfter"
            movej(internos, a=0.6981317007977318, v=0.5235987755982988)
            $ 1645 "Wait: 0.3"
            sleep(0.3)
            $ 1646 "Set CO[1]=Apagar"
            set_configurable_digital_out(1, False)
            $ 1647 "Wait: 0.3"
            sleep(0.3)
            $ 1648 "If barrenoActual≟13"
            if (barrenoActual == 13):
              $ 1649 "Direction: Base Z+"
              global move_thread_flag_1649=0
              thread move_thread_1649():
                enter_critical
                move_thread_flag_1649 = 1
                local towardsPos=calculate_point_to_move_towards(p[0.0,0.0,0.0,0.0,0.0,0.0], [0.0,0.0,1.0], 0.03)
                movel(towardsPos, a=0.04, v=0.03)
                move_thread_flag_1649 = 2
                exit_critical
              end
              move_thread_flag_1649 = 0
              move_thread_han_1649 = run move_thread_1649()
              while (True):
                sleep(1.0E-10)
                if (move_thread_flag_1649 > 1):
                  join move_thread_han_1649
                  $ 1650 "Until (distance)"
                  break
                end
                sync()
              end
              $ 1651 "MoveJ"
              $ 1652 "Zona_der1" "breakAfter"
              movej(get_inverse_kin(Zona_der1_p, qnear=Zona_der1_q), a=1.3962634015954636, v=1.0471975511965976)
              $ 1653 "Posicion_Cero" "breakAfter"
              movej(get_inverse_kin(Posicion_Cero_p, qnear=Posicion_Cero_q), a=1.3962634015954636, v=1.0471975511965976)
              $ 1654 "Call Quitar_Broca_Chida"
              Quitar_Broca_Chida()
              $ 1655 "Call Poner_Broca"
              Poner_Broca()
              $ 1656 "MoveJ"
              $ 1657 "Posicion_Cero" "breakAfter"
              movej(get_inverse_kin(Posicion_Cero_p, qnear=Posicion_Cero_q), a=1.3962634015954636, v=1.0471975511965976)
              $ 1658 "Zona_der1" "breakAfter"
              movej(get_inverse_kin(Zona_der1_p, qnear=Zona_der1_q), a=1.3962634015954636, v=1.0471975511965976)
            else:
              $ 1659 "ElseIf barrenoActual≟27"
              if (barrenoActual == 27):
                $ 1660 "Direction: Base Z+"
                global move_thread_flag_1660=0
                thread move_thread_1660():
                  enter_critical
                  move_thread_flag_1660 = 1
                  local towardsPos=calculate_point_to_move_towards(p[0.0,0.0,0.0,0.0,0.0,0.0], [0.0,0.0,1.0], 0.03)
                  movel(towardsPos, a=0.04, v=0.03)
                  move_thread_flag_1660 = 2
                  exit_critical
                end
                move_thread_flag_1660 = 0
                move_thread_han_1660 = run move_thread_1660()
                while (True):
                  sleep(1.0E-10)
                  if (move_thread_flag_1660 > 1):
                    join move_thread_han_1660
                    $ 1661 "Until (distance)"
                    break
                  end
                  sync()
                end
                $ 1662 "MoveJ"
                $ 1663 "Zona_der1" "breakAfter"
                movej(get_inverse_kin(Zona_der1_p, qnear=Zona_der1_q), a=1.3962634015954636, v=1.0471975511965976)
                $ 1664 "Posicion_Cero" "breakAfter"
                movej(get_inverse_kin(Posicion_Cero_p, qnear=Posicion_Cero_q), a=1.3962634015954636, v=1.0471975511965976)
                $ 1665 "Call Quitar_Broca_Chida"
                Quitar_Broca_Chida()
                $ 1666 "Set carrusel_home=Encender"
                modbus_set_output_signal("carrusel_home", True)
                $ 1667 "Wait: 1.0"
                sleep(1.0)
                $ 1668 "Set carrusel_home=Apagar"
                modbus_set_output_signal("carrusel_home", False)
                $ 1669 "Set mensaje_mw10=120"
                modbus_set_output_register("mensaje_mw10", 120)
                $ 1670 "Wait Continuar_M30=HI"
                while (modbus_get_signal_status("Continuar_M30") == False):
                  sync()
                end
                $ 1671 "Wait: 1.0"
                sleep(1.0)
                $ 1672 "Set mensaje_mw10=100"
                modbus_set_output_register("mensaje_mw10", 100)
                $ 1673 "Wait Continuar_M30=HI"
                while (modbus_get_signal_status("Continuar_M30") == False):
                  sync()
                end
                $ 1674 "Wait: 1.0"
                sleep(1.0)
                $ 1675 "MoveJ"
                $ 1676 "Traslacion_der" "breakAfter"
                movej(get_inverse_kin(Traslacion_der_p, qnear=Traslacion_der_q), a=1.3962634015954636, v=1.0471975511965976)
              end
            end
            $ 1677 "barrenoActual≔barrenoActual+1"
            global barrenoActual=barrenoActual+1
          end
          $ 1678 "Set pos4_term_m612=Encender"
          modbus_set_output_signal("pos4_term_m612", True)
          $ 1679 "Wait: 1.0"
          sleep(1.0)
          $ 1680 "Set pos4_term_m612=Apagar"
          modbus_set_output_signal("pos4_term_m612", False)
        end
      end
      $ 1786 "Traslacion"
      $ 1787 "MoveJ"
      $ 1788 "Traslacion_der" "breakAfter"
      movej(get_inverse_kin(Traslacion_der_p, qnear=Traslacion_der_q), a=1.3962634015954636, v=1.0471975511965976)
      $ 1789 "Set mensaje_mw10=105"
      modbus_set_output_register("mensaje_mw10", 105)
      $ 1790 "Wait Continuar_M30=HI"
      while (modbus_get_signal_status("Continuar_M30") == False):
        sync()
      end
      $ 1791 "Wait: 1.0"
      sleep(1.0)
      $ 1792 "Set mensaje_mw10=110"
      modbus_set_output_register("mensaje_mw10", 110)
      $ 1793 "Wait Continuar_M30=HI"
      while (modbus_get_signal_status("Continuar_M30") == False):
        sync()
      end
      $ 1794 "Wait: 1.0"
      sleep(1.0)
      $ 1795 "Set postrnas_m187=Encender"
      modbus_set_output_signal("postrnas_m187", True)
      $ 1796 "Wait: 1.0"
      sleep(1.0)
      $ 1797 "Set Home_M20=Encender"
      modbus_set_output_signal("Home_M20", True)
      $ 1798 "Wait: 1.0"
      sleep(1.0)
      $ 1799 "Set Home_M20=Apagar"
      modbus_set_output_signal("Home_M20", False)
      $ 1800 "Set postrnas_m187=Apagar"
      modbus_set_output_signal("postrnas_m187", False)
      $ 1801 "Wait: 10.0"
      sleep(10.0)
      $ 1802 "Apagar"
      $ 1803 "Set mensaje_mw10=115"
      modbus_set_output_register("mensaje_mw10", 115)
      $ 1804 "Wait Continuar_M30=HI"
      while (modbus_get_signal_status("Continuar_M30") == False):
        sync()
      end
      $ 1805 "Wait: 1.0"
      sleep(1.0)
      $ 1806 "MoveJ"
      $ 1807 "Waypoint_8" "breakAfter"
      movej(get_inverse_kin(Waypoint_8_p, qnear=Waypoint_8_q), a=1.3962634015954636, v=1.0471975511965976)
      $ 1808 "Off_derecha" "breakAfter"
      movej(get_inverse_kin(Off_derecha_p, qnear=Off_derecha_q), a=1.3962634015954636, v=1.0471975511965976)
      $ 1809 "Set mensaje_mw10=0"
      modbus_set_output_register("mensaje_mw10", 0)
      $ 1810 "Wait: 1.0"
      sleep(1.0)
      $ 1811 "Wait Continuar_M30=HI"
      while (modbus_get_signal_status("Continuar_M30") == False):
        sync()
      end
      $ 1812 "Wait: 1.0"
      sleep(1.0)
      $ 1813 "Popup: Apagar DAS"
      popup("Apagar DAS", "Advertencia", True, False, blocking=False)
      halt
    else:
      $ 1814 "ElseIf Lado_Correr≟1"
      if (modbus_get_signal_status("Lado_Correr") == 1):
        $ 1815 "Set mensaje_mw10=205"
        modbus_set_output_register("mensaje_mw10", 205)
      else:
        $ 1816 "ElseIf Lado_Correr≟0"
        if (modbus_get_signal_status("Lado_Correr") == 0):
          $ 1817 "Set mensaje_mw10=205"
          modbus_set_output_register("mensaje_mw10", 205)
        else:
          $ 1818 "Else" "noBreak"
          $ 1819 "Lado≔ False "
          global Lado=  False
          $ 1820 "Set mensaje_mw10=205"
          modbus_set_output_register("mensaje_mw10", 205)
          $ 1821 "Popup: DAS no anclado"
          popup("DAS no anclado", "Advertencia", True, False, blocking=False)
          halt
        end
      end
    end
  end
end
